/// Rolling interval to create a new log file when expired. 
{attribute 'qualified_only'}
{attribute 'strict'}
{attrivute 'to_string'}
TYPE RollingInterval :
(
	None := 0,
	Hourly,
	Daily,
	Monthly
);
END_TYPE

(* stored: Version 1.1.0.1
   DUT RollingInterval: Id {6307f971-7bf8-46ec-9b38-ec512e24283a} *)
